TYPE ST_CanQueue :
STRUCT
	TxCounter : UINT;
	RxCounter : UINT;
	NoOfMessages : UINT;
	Messages : ARRAY[0..(GVL_ODrive.nMaxMsgCount-1)] OF ST_CanMessage;	// Message length should according to io device setting
END_STRUCT
END_TYPE

(* stored: Version 1.1.0.1
   DUT ST_CanQueue: Id {75b2d68c-ca7f-46e4-a091-39a52f8b73b3} *)
